PROGRAM PILS_DEVICES
VAR
END_VAR

//Interface between PILS and AXIS
//Example code of how to link the axis and PILS
fbMotorM1(stAxisStruct:= astAxes[1], stDeviceStructPILS:= stMotorM1, stAxisPar:= stMotorM1Param);
fbMotorM2(stAxisStruct:= astAxes[2], stDeviceStructPILS:= stMotorM2, stAxisPar:= stMotorM2Param);
stPowerSwitchesAxis1.nValue:= BOOL_TO_INT(Axis_Template.bPowerSwitchesAxis1);
stPowerSwitchesAxis2.nValue:= BOOL_TO_INT(Axis_Template.bPowerSwitchesAxis2);
//stPowerSwitchesAxis1Ctr.nCurrentValue:= BOOL_TO_INT(Axis_Template.bPowerSwitchesAxis1);
//stPowerSwitchesAxis1Ctr.nTargetValue:= BOOL_TO_INT(Axis_Template.bPowerSwitchesAxis1);

//stMotor1Temp.fValue := Axis_1.fMotTemp1;
//stMotorM1EncoderRaw.nValue := nEncoderValueAxis1;

END_PROGRAM

(* stored: Version 1.1.0.1, ProductVersion 3.1.4024.10
   POU PILS_DEVICES: Id {c13d0ec1-dadc-4beb-a3f1-3a752770c4f8}, SpecialFunc None *)
